//==================================================================================================
//							Beckhoff Automation Poland
//									25.04.2018
//		Program obslugujacy pamiec nieulotna 
//	v1.4    || TC v 3.1.4026.19		|| - Obsługa UPS
// 	v1.3	|| TC v 3.1.4022.16		|| - Przeniesienie logowania do EvenLogger'a do programu P_SystemDiag_EventLog
// 	v1.2	|| TC v 3.1.4022.0		|| - Dodanie akcji UPS
//	v1.1 	|| TC v 3.1.4020.14 	|| - Dodane wyjscia bOk, bWarning, bError
//	v1.0 	|| TC v 3.1.4020.0 		|| - Pierwsza wersja
//==================================================================================================
PROGRAM P_Persistent
VAR_INPUT
	sAmsNetID_EtherCATMaster	: T_AmsNetId	:= '192.168.40.160.3.1';			// EtherCAT Master AMS Net ID
	bWritePersistent			: BOOL;
	bReset						: BOOL;
END_VAR
VAR_OUTPUT
	bOK							: BOOL 						:= TRUE;				// Brak bledow i ostrzezen
	bWarning					: BOOL;												// Ostrzezenie
	bError						: BOOL;												// Zbiorcza flaga bledow
	udiErrorID					: UDINT;
	sErrorDescription			: WSTRING;
	bWrited						: BOOL;
	bPowerFailDetect			: BOOL;
END_VAR
VAR																			
	iStep						: INT;
	fbWritePersistentData		: FB_WritePersistentData;
	
	//fbUPS						: FB_S_UPS;
	//fbUPS_CB3011				: FB_S_UPS_CB3011;
	fbUPS_CX51x0				: FB_S_UPS_CX51x0;
	//fbUPS_CX9020_U900			: FB_S_UPS_CX9020_U900;
	//fbUPS_BAPI					: FB_S_UPS_BAPI;
	fbUPS_CU8130				:FB_GetUPSStatus;
	
	eUpsMode					: E_S_UPS_Mode;
	eUpsState					: E_S_UPS_State;
	
	
	iNumberOfWrites				: INT;
	rtWritePersistent			: R_TRIG;
END_VAR


ACT_UPS();
ACT_WritePersistent();

fbUPS_CU8130.stStatus.ePowerStatus;
fbUPS_CU8130.stStatus.eBatteryStatus;
fbUPS_CU8130.stStatus.nPowerFailCnt;
fbUPS_CU8130.stStatus.eCommStatus;
IF fbUPS_CU8130.stStatus.ePowerStatus=2 AND NOT bWrited THEN
	bWritePersistent:=TRUE;
ELSE
	bWritePersistent:=FALSE;
END_IF

ACTION A_fbS_UPS:
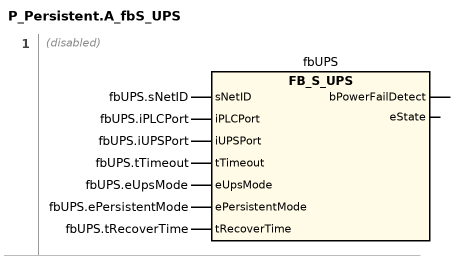
// NETWORK 1 (disabled)
// fbUPS(
//     sNetID := fbUPS.sNetID,
//     iPLCPort := fbUPS.iPLCPort,
//     iUPSPort := fbUPS.iUPSPort,
//     tTimeout := fbUPS.tTimeout,
//     eUpsMode := fbUPS.eUpsMode,
//     ePersistentMode := fbUPS.ePersistentMode,
//     tRecoverTime := fbUPS.tRecoverTime); // FB_S_UPS
END_ACTION

ACTION A_fbS_UPS_BAPI:
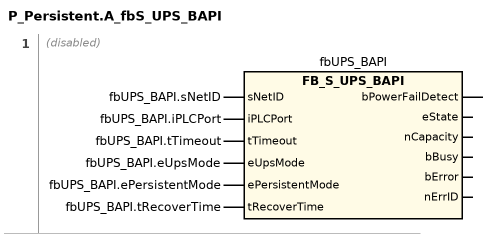
// NETWORK 1 (disabled)
// fbUPS_BAPI(
//     sNetID := fbUPS_BAPI.sNetID,
//     iPLCPort := fbUPS_BAPI.iPLCPort,
//     tTimeout := fbUPS_BAPI.tTimeout,
//     eUpsMode := fbUPS_BAPI.eUpsMode,
//     ePersistentMode := fbUPS_BAPI.ePersistentMode,
//     tRecoverTime := fbUPS_BAPI.tRecoverTime); // FB_S_UPS_BAPI
END_ACTION

ACTION A_fbS_UPS_CB3011:
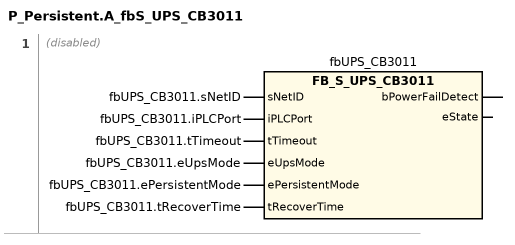
// NETWORK 1 (disabled)
// fbUPS_CB3011(
//     sNetID := fbUPS_CB3011.sNetID,
//     iPLCPort := fbUPS_CB3011.iPLCPort,
//     tTimeout := fbUPS_CB3011.tTimeout,
//     eUpsMode := fbUPS_CB3011.eUpsMode,
//     ePersistentMode := fbUPS_CB3011.ePersistentMode,
//     tRecoverTime := fbUPS_CB3011.tRecoverTime); // FB_S_UPS_CB3011
END_ACTION

ACTION A_fbS_UPS_CX51x0:
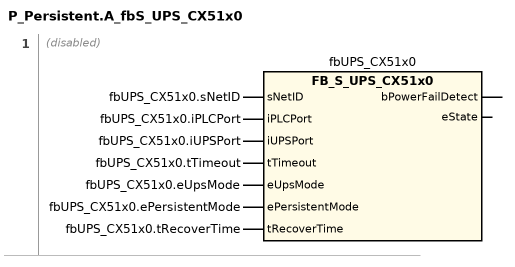
// NETWORK 1 (disabled)
// fbUPS_CX51x0(
//     sNetID := fbUPS_CX51x0.sNetID,
//     iPLCPort := fbUPS_CX51x0.iPLCPort,
//     iUPSPort := fbUPS_CX51x0.iUPSPort,
//     tTimeout := fbUPS_CX51x0.tTimeout,
//     eUpsMode := fbUPS_CX51x0.eUpsMode,
//     ePersistentMode := fbUPS_CX51x0.ePersistentMode,
//     tRecoverTime := fbUPS_CX51x0.tRecoverTime); // FB_S_UPS_CX51x0
END_ACTION

ACTION A_fbS_UPS_CX9020_U900:
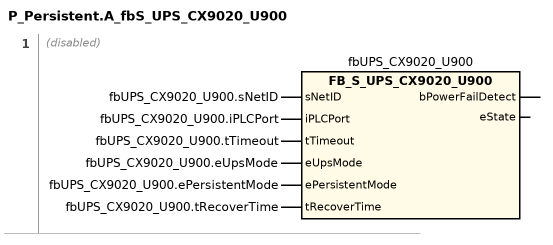
// NETWORK 1 (disabled)
// fbUPS_CX9020_U900(
//     sNetID := fbUPS_CX9020_U900.sNetID,
//     iPLCPort := fbUPS_CX9020_U900.iPLCPort,
//     tTimeout := fbUPS_CX9020_U900.tTimeout,
//     eUpsMode := fbUPS_CX9020_U900.eUpsMode,
//     ePersistentMode := fbUPS_CX9020_U900.ePersistentMode,
//     tRecoverTime := fbUPS_CX9020_U900.tRecoverTime); // FB_S_UPS_CX9020_U900
END_ACTION

ACTION ACT_UPS:
//fbUPS_CX9020_U900
//(
//	sNetID							:= sAmsNetID_EtherCATMaster, 
//	iPLCPort						:= 851, 
//	tTimeout						:= DEFAULT_ADS_TIMEOUT, 
//	eUpsMode						:= E_S_UPS_Mode.eSUPS_WrPersistData_Shutdown,
//	ePersistentMode					:= E_PersistentMode.SPDM_2PASS, 
//	tRecoverTime					:= T#10S, 
//	bPowerFailDetect				=> bPowerFailDetect, 
//	eState							=> eUpsState
//);


//fbUPS_CX51x0
//(
//	sNetID							:= sAmsNetID_EtherCATMaster, 
//	iPLCPort						:= 851, 
//	iUPSPort						:= 16#588, 
//	tTimeout						:= DEFAULT_ADS_TIMEOUT, 
//	eUpsMode						:= E_S_UPS_Mode.eSUPS_WrPersistData_Shutdown, 
//	ePersistentMode					:= E_PersistentMode.SPDM_2PASS, 
//	tRecoverTime					:= T#10S, 
//	bPowerFailDetect				=> bPowerFailDetect, 
//	eState							=> eUpsState
//);
fbUPS_CU8130
(	sNetID							:='',
	nPort							:=0,
	bEnable							:=TRUE,
	bValid							=>,
	bError	=>,
	nErrId =>,
	stStatus =>,);
END_ACTION

ACTION ACT_WritePersistent:
rtWritePersistent(CLK:= bWritePersistent);


CASE iStep OF

0:
	IF rtWritePersistent.Q THEN
		fbWritePersistentData.PORT												:= _AppInfo.AdsPort;
		fbWritePersistentData.MODE												:= SPDM_2PASS;	
		fbWritePersistentData.START												:= TRUE;
		bWrited																	:= FALSE;
		iStep:= 10;
	END_IF

10:
	IF NOT fbWritePersistentData.BUSY THEN
		IF NOT fbWritePersistentData.ERR THEN
			fbWritePersistentData.START											:= FALSE;
			bWrited																:= TRUE;	
			iNumberOfWrites														:= iNumberOfWrites + 1;
			iStep:= 20;
		END_IF
	END_IF

	IF fbWritePersistentData.ERR THEN
 	
		bWrited																	:= FALSE;
		bError																	:= TRUE;	
		udiErrorID																:= fbWritePersistentData.ERRID;
		sErrorDescription														:= "Błąd zapisu zmiennych PERSISTENT";
		iStep:= 900;
	END_IF
	
20:
	IF NOT bWritePersistent THEN
		iStep:= 0;
	END_IF	
	
900:
	bOK																			:= FALSE;
	
	IF bReset THEN
		fbWritePersistentData.START												:= FALSE;
	END_IF
	IF NOT bReset THEN
		fbWritePersistentData.START												:= TRUE;
	END_IF
	
	
	IF NOT fbWritePersistentData.BUSY THEN
		IF NOT fbWritePersistentData.ERR THEN 
			bOK																	:= TRUE;
			bError																:= FALSE;
			udiErrorID															:= 0;
			sErrorDescription													:= "";
			iStep:= 0;	
		END_IF
	END_IF
	

END_CASE


fbWritePersistentData();
END_ACTION

END_PROGRAM

(* stored: Version 1.1.0.1, ProductVersion 3.1.4026.13, FileIdentifier d6f6be2ebd6c0005a070eeec2b23fdef0b6df8f9, FileSignature 7f15dda74d59e3e5551b6920e9b94a6c84a75bfb6c2924c7629182631389966810f3a61d98d065b770a948dff155cd8d76a401fdf686f7598cb5beaf933adc6f2f719bebc03947b483e9c4a212c57d01a034adeb7b500fe495b3a7a695309bb8d3b6755915e1a2500e19f5349d16b148d77f5b75d8e5c49a46e4ca839c2914f386a835ff648347159946b2206cedbd0a098f3a6fbd98134c19372c3ebd72470e958bfb03a556f3f56ef928e53f60ef6a885a61510157066b2da568c1d76bc47c450741bca965913cae0c328d4414494baf0a19f63c298024a1e97cb855eb50713a11f096610168cf09f407d46f0194db19d4c6fc1ad06928a7902ddf652fc5b7
   POU P_Persistent: Id {188d73a3-0452-479f-b48c-0ee7551b4de1}, SpecialFunc None
   Folder NotUsed: Id {5bcd16f8-baa0-449f-bea0-e4f57b54dbc7}
   Action A_fbS_UPS: Id {8b222a48-c306-4706-9d37-e32da7b93a34}
   Action A_fbS_UPS_BAPI: Id {af48fac2-ce8b-4607-8e0a-49a7299bcf3a}
   Action A_fbS_UPS_CB3011: Id {4240ce2d-4cb7-49af-8c56-ac9a76010f70}
   Action A_fbS_UPS_CX51x0: Id {88db6106-cabd-4b4c-b4f8-cd49e3cad3b2}
   Action A_fbS_UPS_CX9020_U900: Id {b44081b3-05fd-45ca-8206-461be1a03847}
   Action ACT_UPS: Id {a63f71ea-cd18-4c5b-8ecd-5a9783d20bb5}
   Action ACT_WritePersistent: Id {ce0926f9-4d7d-4eac-a9af-4a2692fa7350} *)
